FUNCTION_BLOCK _BIT_UsingMockStructure_TestSuite EXTENDS TcUnit.FB_TestSuite
VAR
END_VAR

TestAddress();
TestClearReference();
TestClone();
TestTypeNameReturnsExpected();
TestMakeReferenceToFollowsReference();
TestMakeReferenceToUpdatesReference();
TestSize();
TestValueReturnsExpectedAfterChange();
TestSerializeTypeWith();
TestSerializeWith();
TestTryDeserializeFrom();
TestTryMakeReferenceToFollowsReference();
TestTryMakeReferenceToUpdatesReference();

METHOD PUBLIC TestAddress
VAR
    _type : _MyStruct;
    notExpected : PVOID := 0;
    actual : PVOID;
END_VAR
TEST('TestAddress');

actual := _type.MyBit.Address;

AssertFalse(
    Condition := (notExpected = actual),
    Message := 'Type did not return a valid address.'
);

TEST_FINISHED();
END_METHOD

METHOD PUBLIC TestClearReference
VAR
    _type : _MyStruct;
	target : MyStruct;
    expected : BOOL := FALSE;
    actual : BOOL;
END_VAR
TEST('TestClearReference');

_type.MakeReferenceTo(target);
_type.ClearReference();
target.MyBit := TRUE;

actual := _type.MyBit.Value;

AssertEquals(
    Expected := expected,
    Actual := actual,
    Message := 'Value incorrectly followed target change'
);

TEST_FINISHED();
END_METHOD

METHOD PUBLIC TestClone
VAR
    _type : _MyStruct;
	clone : I_Datatype;
	isValidClone : BOOL;
	compareResult : DINT;
END_VAR
TEST('TestClone');

clone := _type.Clone();

isValidClone := clone <> 0;

IF isValidClone THEN
	compareResult := memcmp(_type.Address, clone.Address, clone.Size);
END_IF

AssertTrue(
	Condition := isValidClone,
	Message := 'Clone did not produce a clone'
);

clone.Dispose();

TEST_FINISHED();
END_METHOD

METHOD PUBLIC TestMakeReferenceToFollowsReference
VAR
    _type : _MyStruct;
	target : MyStruct;
    expected : BOOL := TRUE;
    actual : BOOL;
END_VAR
TEST('TestMakeReferenceToFollowsReference');

_type.MakeReferenceTo(target);
target.MyBit := TRUE;

actual := _type.MyBit.Value;

AssertEquals(
    Expected := expected,
    Actual := actual,
    Message := 'Value did not follow target change'
);

TEST_FINISHED();
END_METHOD

METHOD PUBLIC TestMakeReferenceToUpdatesReference
VAR
    _type : _MyStruct;
	target : MyStruct;
    expected : BOOL := TRUE;
    actual : BOOL;
END_VAR
TEST('TestMakeReferenceToUpdatesReference');

_type.MakeReferenceTo(target);
_type.MyBit.Value:= TRUE;

actual := target.MyBit;

AssertEquals(
    Expected := expected,
    Actual := actual,
    Message := 'Value did not update target'
);

TEST_FINISHED();
END_METHOD

METHOD PUBLIC TestSerializeTypeWith
VAR
    _type : _MyStruct;
    serializer : JsonSerializer;
    expected : STRING := '{"typeName":"BIT"}';
    actual : STRING(500);
END_VAR
TEST('TestSerializeTypeWith');

serializer.Reset();
_type.MyBit.SerializeTypeWith(serializer);
serializer.TryGetSerializedData(ADR(actual), SIZEOF(actual));

AssertEquals_STRING(
    Expected := expected,
    Actual := actual,
    Message := 'Serialization of type did not return correct string.'
);

TEST_FINISHED();
END_METHOD

METHOD PUBLIC TestSerializeWith
VAR
    _type : _MyStruct;
    serializer : JsonSerializer;
    expected : STRING := 'true';
    actual : STRING(500);
END_VAR
TEST('TestSerializeWith');

serializer.Reset();
_type.MyBit.Value := true;
_type.MyBit.SerializeWith(serializer);
serializer.TryGetSerializedData(ADR(actual), SIZEOF(actual));

AssertEquals_STRING(
    Expected := expected,
    Actual := actual,
    Message := 'Serialization of type data did not return correct string.'
);

TEST_FINISHED();
END_METHOD

METHOD PUBLIC TestSize
VAR
    _type : _MyStruct;
    expected : UDINT := SIZEOF(MyStruct.MyBit);
    actual : UDINT;
END_VAR
TEST('TestSize');

actual := _type.MyBit.Size;

AssertEquals_UDINT(
    Expected := Expected,
    Actual := actual,
    Message := 'Type did not return the correct size.'
);

TEST_FINISHED();
END_METHOD

METHOD PUBLIC TestTryDeserializeFrom
VAR
    deserializer : JsonDeserializer;
    feedback : DeserializerFeedback;
    json : STRING := 'true';
    _type : _MyStruct;
    expected : BOOL := TRUE;
    actual : BOOL;
 END_VAR
TEST('TestTryDeserializeFrom');

deserializer.Reset();
deserializer.TryLoad(json);
_type.MyBit.TryDeserializeFrom(Deserializer, Feedback);

actual := _type.MyBit.Value;

AssertEquals(
    Expected := expected,
    Actual := actual,
    Message := 'Type did not deserialize correctly.'
);

TEST_FINISHED();
END_METHOD

METHOD PUBLIC TestTryMakeReferenceToFollowsReference
VAR
    _type : _MyStruct;
	target : _MyStruct;
    expected : BOOL := TRUE;
    actual : BOOL;
END_VAR
TEST('TestTryMakeReferenceToFollowsReference');

_type.TryMakeReferenceTo(target);
target.MyBit.Value := TRUE;

actual := _type.MyBit.Value;

AssertEquals(
    Expected := expected,
    Actual := actual,
    Message := 'Value did not follow target change'
);

TEST_FINISHED();
END_METHOD

METHOD PUBLIC TestTryMakeReferenceToUpdatesReference
VAR
    _type : _MyStruct;
	target : _MyStruct;
    expected : BOOL := TRUE;
    actual : BOOL;
END_VAR
TEST('TestTryMakeReferenceToUpdatesReference');

_type.TryMakeReferenceTo(target);
_type.MyBit.Value := TRUE;

actual := target.MyBit.Value;

AssertEquals(
    Expected := expected,
    Actual := actual,
    Message := 'Value did not update target'
);

TEST_FINISHED();
END_METHOD

METHOD PUBLIC TestTypeNameReturnsExpected
VAR
    _type : _MyStruct;
    expected : STRING := 'BIT';
    actual : STRING;
END_VAR
TEST('TestTypeNameReturnsExpected');

actual := _type.MyBit.TypeName;

AssertEquals_STRING(
    Expected := expected,
    Actual := actual,
    Message := 'Type did not return correct iec type.'
);

TEST_FINISHED();
END_METHOD

METHOD PUBLIC TestValueReturnsExpectedAfterChange
VAR
    _type : _MyStruct;
    expected : BOOL := FALSE;
    actual : BOOL;
END_VAR
TEST('TestValueReturnsExpectedAfterChange');

_type.MyBit.Value := FALSE;

actual := _type.MyBit.Value;

AssertEquals(
    Expected := expected,
    Actual := actual,
    Message := 'Expected value not returned after change.'
);

TEST_FINISHED();
END_METHOD

END_FUNCTION_BLOCK

(* stored: Version 1.1.0.1, ProductVersion 3.1.4024.12
   POU _BIT_UsingMockStructure_TestSuite: Id {53776d77-cd69-4cba-a501-6062c9c4573c}, SpecialFunc None
   Method TestAddress: Id {1d27ee1f-0b09-4785-b8d2-bcd3ab86453c}
   Method TestClearReference: Id {3435f573-ddcd-429a-990f-ab9da5a59bfe}
   Method TestClone: Id {4c2de117-d9d9-4cc0-95cb-a8fe2089f37a}
   Method TestMakeReferenceToFollowsReference: Id {3a249014-86e0-498f-9722-53979105fbeb}
   Method TestMakeReferenceToUpdatesReference: Id {3b11cd5f-8741-4890-b67e-414d5a8c0cf4}
   Method TestSerializeTypeWith: Id {797c5fd7-fd19-400d-a960-ccee07865a82}
   Method TestSerializeWith: Id {60d8f49a-4c82-44d2-854b-1fad461a0e43}
   Method TestSize: Id {564cfc4b-7d54-451e-bac5-159dd61fd000}
   Method TestTryDeserializeFrom: Id {4c4d66a3-bdce-4d50-bda3-28c5daf2940b}
   Method TestTryMakeReferenceToFollowsReference: Id {0ca366a1-c314-4171-b7bf-dc92fcc4fdd4}
   Method TestTryMakeReferenceToUpdatesReference: Id {da0494dc-0edf-45cb-bcf0-34362e28786e}
   Method TestTypeNameReturnsExpected: Id {a423b94b-4bbe-43e3-b0d7-6b0eea2a41c9}
   Method TestValueReturnsExpectedAfterChange: Id {7e4f43c9-8cd1-4886-8829-6d31fb64643e} *)
